// Mitsubishi GX Works2 project: 230927-003-or   PLC: Q03UDV

// task Task_01 (event TRUE, interval 0, priority 31): POU_01

PROGRAM POU_01
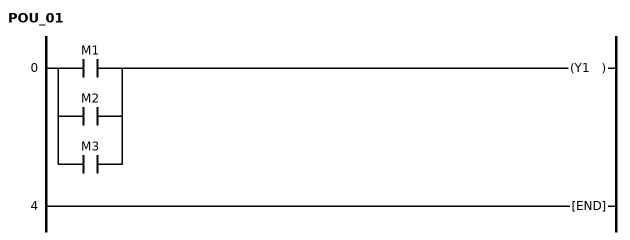
0     LD      M1
      OR      M2
      OR      M3
      OUT     Y1
4     END
END_PROGRAM
